// TIA Portal V17 export
// export: Created 2025-03-10T13:12:42.778462Z, ExportSetting WithDefaults, DisplayName Totally Integrated Automation Portal, DisplayVersion V17 Update 8, DisplayName TIA Portal Openness, DisplayVersion V17 Update 8, DisplayName TIA Portal Version Control Interface, DisplayVersion V17, DisplayName SINAMICS Startdrive Advanced, DisplayVersion V17 SP2, DisplayName SINAMICS Startdrive G110M, G120, G120C, G120D, G120P, G115D, DisplayVersion V17 SP2, DisplayName SINAMICS Startdrive G130, G150, S120, S150, SINAMICS MV, S210, DisplayVersion V17 SP2, DisplayName STEP 7 Professional, DisplayVersion V17 Update 8, DisplayName SINUMERIK ONE STEP 7 Toolbox, DisplayVersion V17 Update 12, DisplayName SINUMERIK 840D sl STEP 7 Toolbox, DisplayVersion V17 Update 12, DisplayName STEP 7 Safety, DisplayVersion V17 Update 6, DisplayName WinCC Advanced, DisplayVersion V17 Update 8
DATA_BLOCK "DB2041_WINCC_HMI_LINES_STATIONS"   // DB2041
{ S7_Optimized_Access := 'FALSE'; DB_Accessible_From_OPC_UA := 'FALSE' }
AUTHOR : ETXETAR
VERSION : 1.0
// stored: AutoNumber false, DBAccessibleFromOPCUA false, DBAccessibleFromWebserver true, IsOnlyStoredInLoadMemory false, IsWriteProtectedInAS false
   VAR RETAIN
      STATION_1 { S7_SetPoint := 'True'} : Array[1..20] of "WINCC_HMI_LINES";
      STATION_2 { S7_SetPoint := 'True'} : Array[1..20] of "WINCC_HMI_LINES";
      STATION_3 { S7_SetPoint := 'True'} : Array[1..20] of "WINCC_HMI_LINES";
      STATION_4 { S7_SetPoint := 'True'} : Array[1..20] of "WINCC_HMI_LINES";
      STATION_5 { S7_SetPoint := 'True'} : Array[1..20] of "WINCC_HMI_LINES";
      STATION_6 { S7_SetPoint := 'True'} : Array[1..20] of "WINCC_HMI_LINES";
      STATION_7 { S7_SetPoint := 'True'} : Array[1..20] of "WINCC_HMI_LINES";
      STATION_8 { S7_SetPoint := 'True'} : Array[1..20] of "WINCC_HMI_LINES";
      STATION_9 { S7_SetPoint := 'True'} : Array[1..20] of "WINCC_HMI_LINES";
      STATION_10 { S7_SetPoint := 'True'} : Array[1..20] of "WINCC_HMI_LINES";
   END_VAR
BEGIN
END_DATA_BLOCK
